// TIA Portal project "MachacaderaAridos" (V16)

(* hardware
DEVICE "S7-1200 station_1"  S7-1200 Station
   slot 0: "Rack_0"  S7-1200 Rack  Rack  V1.0
   slot 1: "PLC_1"  CPU 1214C AC/DC/Rly  6ES7 214-1BG40-0XB0  V4.2
   slot 3: "DQ 4x24VDC_1"  DQ4 signal board (200 kHz)  6ES7 222-1BD30-0XB0  V1.0
*)

// ===== PLC "PLC_1"  CPU 1214C AC/DC/Rly =====

VAR_GLOBAL   // PLC tag table "Entradas"
   "Interruptor de Marcha" AT %I0.4 : Bool;
   "Relé Térmico Motor1" AT %I0.1 : Bool;
   "Relé Térmico Motor2" AT %I0.2 : Bool;
   "Relé Térmico Motor3" AT %I0.3 : Bool;
   "Relé Sobrecarga M2" AT %I0.0 : Bool;
END_VAR

VAR_GLOBAL   // PLC tag table "Salidas"
   "Contactor Motor M1" AT %Q0.0 : Bool;
   "Contactor Motor M2" AT %Q0.1 : Bool;
   "Contactor Motor M3" AT %Q0.2 : Bool;
   "Alarma" AT %Q0.3 : Bool;
END_VAR

ORGANIZATION_BLOCK "Main"   // OB1, LAD, ProgramCycle
TITLE = "Main Program Sweep (Cycle)"
{ S7_Optimized_Access := 'TRUE' }
VERSION : 0.1
   VAR_INPUT
      Initial_Call : Bool;   // Initial call of this OB
      Remanence : Bool;   // =True, if remanent data are available
   END_VAR
BEGIN

REGION Network 1
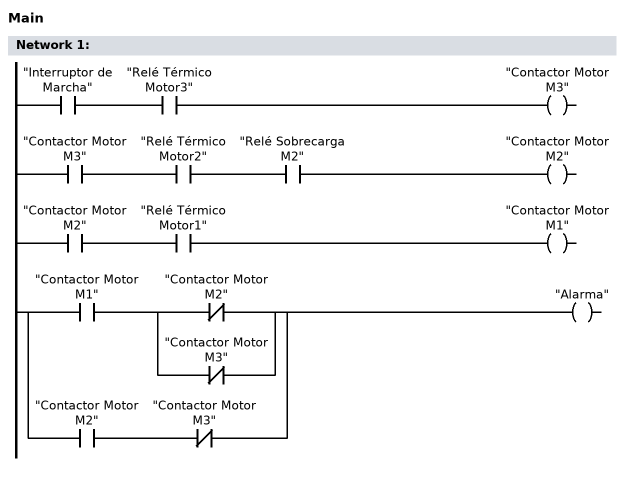
   RUNG wire#powerrail
      Contact( "Interruptor de Marcha" )
      Contact( "Relé Térmico Motor3" )
      Coil( "Contactor Motor M3" )
   END_RUNG
   RUNG wire#powerrail
      Contact( "Contactor Motor M3" )
      Contact( "Relé Térmico Motor2" )
      Contact( "Relé Sobrecarga M2" )
      Coil( "Contactor Motor M2" )
   END_RUNG
   RUNG wire#powerrail
      Contact( "Contactor Motor M2" )
      Contact( "Relé Térmico Motor1" )
      Coil( "Contactor Motor M1" )
   END_RUNG
   RUNG wire#powerrail
      Contact( "Contactor Motor M1" )
      wire#w1
      I_Contact( "Contactor Motor M2" )
      wire#w2
      Coil( "Alarma" )
   END_RUNG
   RUNG wire#w1
      I_Contact( "Contactor Motor M3" )
   END_RUNG wire#w2
   RUNG wire#powerrail
      Contact( "Contactor Motor M2" )
      I_Contact( "Contactor Motor M3" )
   END_RUNG wire#w2
   // the same network as SCL:
   "Contactor Motor M3" := "Interruptor de Marcha" AND "Relé Térmico Motor3";
   "Contactor Motor M2" := "Contactor Motor M3" AND "Relé Térmico Motor2" AND "Relé Sobrecarga M2";
   "Contactor Motor M1" := "Contactor Motor M2" AND "Relé Térmico Motor1";
   "Alarma" := ("Contactor Motor M1" AND (NOT "Contactor Motor M2" OR NOT "Contactor Motor M3")) OR ("Contactor Motor M2" AND NOT "Contactor Motor M3");
END_REGION
END_ORGANIZATION_BLOCK